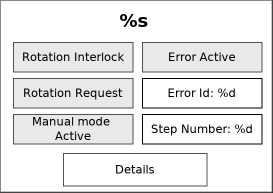
VISUALIZATION vTableBaseStation  // 273x193
VAR_IN_OUT
	fbStation:FB_BaseStation;
	fbTableControl: FB_TableControl;
END_VAR
    Rectangle (0,0 273x193)
    Rectangle (13,78 120x30), "Rotation Request", colour toggle: fbStation.bRotationRequest
    Rectangle (13,42 120x30), "Rotation Interlock", colour toggle: fbStation.bRotationInterlock
    Rectangle (142,42 120x30), "Error Active", colour toggle: fbStation.bError
    Rectangle (13,114 120x30), "Manual mode Active", colour toggle: fbStation.bManualModeActive
    Rectangle (142,78 120x30), "Error Id: %d", text variable: fbStation.udiErrorNumber
    Rectangle (142,114 120x30), "Step Number: %d", text variable: fbStation.iWorkStep
    Rectangle (63,153 144x33), "Details"
        OnMouseDown: execute { fbTableControl.stHMI.iDialogNumber := fbStation.iStationId; }
    Rectangle (59,6 150x30), "%s", text variable: fbStation.sStationName
END_VISUALIZATION

(* stored: Version 1.1.0.1, ProductVersion 3.1.4024.15
   Visu vTableBaseStation: Id {05825a14-3c57-4919-8bf9-646486fd8593} *)
